ABB RobotStudio station: Table with target.rsstn

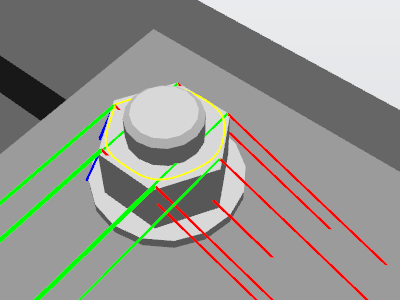
Station Station (saved by RobotStudio 22.3.10141.1)
Controller Controller2
  mechanical unit ROB_1: IRB1410_5_144__01, 6 joints, base frame (0, 0, 0) mm
Layout (positions relative to the parent item):
  - IRB1410_5_144__01 [mechanism, from Robots\IRB1410_5_144_G_01.rslib] at (0, 0, 0) mm; joint values [0.0908, 0.5599, 0.8443, 0.2461, -0.3282, -0.188] (rad or m)
  - table_and_fixture_140 [part, from Training Objects\propeller_table.rslib] at (988.94, -175, 0) mm
  - MyTool [mechanism, from Training Objects\myTool.rslib] at (1105.96, 94, 482.36) mm, rotated rx -180 ry 60 rz -180 deg
Attachment: MyTool is attached to IRB1410_5_144__01 / Link6
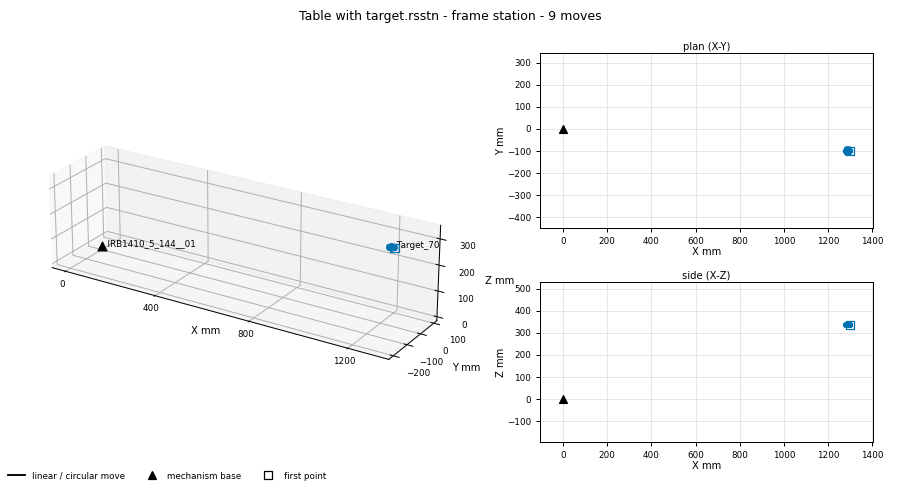
[picture p0: tool path of Table with target.rsstn in frame station, 9 of 9 moves have a stored position in this frame; points joined in program order, loops and branches not executed]
Targets, tools, work objects and paths stored in the station, written as RAPID:
! task T_ROB1
MODULE CalibData
  PERS tooldata MyTool:=[TRUE,[[31.792631019,0,229.638935148],[0.945518576,0,0.325568154,0]],[1,[0,0,1],[1,0,0,0],0,0,0]];
ENDMODULE

! task T_ROB1
MODULE Module1
  CONST robtarget Target_10:=[[1298.606015149,-99.322390924,335.126988795],[0.190805431,0.000000001,0.981627876,0.000000016],[-1,-1,0,0],[9E+09,9E+09,9E+09,9E+09,9E+09,9E+09]];
  CONST robtarget Target_20:=[[1293.833975411,-108.714296883,335.239098516],[0.190804964,0.000000002,0.981627967,0.000000016],[-1,-1,0,0],[9E+09,9E+09,9E+09,9E+09,9E+09,9E+09]];
  CONST robtarget Target_30:=[[1284.016020613,-108.714289941,335.239098112],[0.190804966,0.000000002,0.981627967,0.000000018],[-1,-1,0,0],[9E+09,9E+09,9E+09,9E+09,9E+09,9E+09]];
  CONST robtarget Target_40:=[[1279.428931768,-100.958795352,335.762694702],[0.190804233,-0.000000006,0.981628109,0.000000021],[-1,-1,0,0],[9E+09,9E+09,9E+09,9E+09,9E+09,9E+09]];
  CONST robtarget Target_50:=[[1283.537033031,-91.620253829,335.518813965],[0.190803558,-0.000000004,0.98162824,0.000000021],[-1,-1,0,0],[9E+09,9E+09,9E+09,9E+09,9E+09,9E+09]];
  CONST robtarget Target_60:=[[1294.005032162,-91.620223471,335.518784086],[0.190803449,-0.00000001,0.981628262,0.000000019],[-1,-1,0,0],[9E+09,9E+09,9E+09,9E+09,9E+09,9E+09]];
  CONST robtarget Target_70:=[[1298.231019066,-99.09634302,335.381807422],[0.190802844,-0.000000002,0.981628379,0.000000022],[-1,-1,0,0],[9E+09,9E+09,9E+09,9E+09,9E+09,9E+09]];
  CONST robtarget Target_80:=[[1149.214016226,-99.396362417,334.688483645],[0.190802436,0.000000002,0.981628458,0.00000001],[-1,-1,0,0],[9E+09,9E+09,9E+09,9E+09,9E+09,9E+09]];
  CONST robtarget Target_90:=[[1145.478014256,-109.561191739,336.457915979],[0.190801851,0.000000021,0.981628572,0.000000029],[-1,-1,0,0],[9E+09,9E+09,9E+09,9E+09,9E+09,9E+09]];
  CONST robtarget Target_100:=[[1135.375026076,-109.561186391,336.457899307],[0.190801736,0.000000023,0.981628594,0.000000031],[-1,-1,0,0],[9E+09,9E+09,9E+09,9E+09,9E+09,9E+09]];
  CONST robtarget Target_110:=[[1133.568994915,-109.561194497,334.542287058],[0.190801322,0.000000006,0.981628675,0.000000032],[-1,-1,0,0],[9E+09,9E+09,9E+09,9E+09,9E+09,9E+09]];
  CONST robtarget Target_120:=[[1127.742071524,-109.561197718,324.034410923],[0.190801162,-0.000000004,0.981628706,0.000000029],[-1,-1,0,0],[9E+09,9E+09,9E+09,9E+09,9E+09,9E+09]];
  CONST robtarget Target_130:=[[1132.673969986,-109.561195422,311.197484975],[0.190800844,-0.000000005,0.981628768,0.000000029],[-1,-1,0,0],[9E+09,9E+09,9E+09,9E+09,9E+09,9E+09]];
  CONST robtarget Target_140:=[[1145.380019716,-109.561193614,311.197478936],[0.190800742,-0.000000004,0.981628788,0.000000031],[-1,-1,0,0],[9E+09,9E+09,9E+09,9E+09,9E+09,9E+09]];
  CONST robtarget Target_150:=[[1144.973996719,91.276514259,335.160802204],[0.19080037,-0.000000004,0.98162886,0.000000025],[0,0,-1,0],[9E+09,9E+09,9E+09,9E+09,9E+09,9E+09]];
  CONST robtarget Target_160:=[[1144.973996719,91.276514259,335.160802204],[0.19080037,-0.000000004,0.98162886,0.000000025],[0,0,-1,0],[9E+09,9E+09,9E+09,9E+09,9E+09,9E+09]];
  CONST robtarget Target_170:=[[1144.973996719,91.276514259,335.160802204],[0.19080037,-0.000000004,0.98162886,0.000000025],[0,0,-1,0],[9E+09,9E+09,9E+09,9E+09,9E+09,9E+09]];
  CONST robtarget Target_180:=[[1128.543957252,99.999996916,334.999995635],[0.190800354,-0.000000004,0.981628863,0.000000023],[0,0,-1,0],[9E+09,9E+09,9E+09,9E+09,9E+09,9E+09]];
  CONST robtarget Target_190:=[[1133.739957557,108.999993345,335.000022744],[0.190800372,-0.000000004,0.98162886,0.000000023],[0,0,-1,0],[9E+09,9E+09,9E+09,9E+09,9E+09,9E+09]];
  CONST robtarget Target_200:=[[1144.935946559,99.999995513,322.999995269],[0.190800348,-0.000000005,0.981628864,0.00000002],[0,0,-1,0],[9E+09,9E+09,9E+09,9E+09,9E+09,9E+09]];
  CONST robtarget Target_210:=[[1144.935946559,99.999995513,322.999995269],[0.190800348,-0.000000005,0.981628864,0.00000002],[0,0,-1,0],[9E+09,9E+09,9E+09,9E+09,9E+09,9E+09]];
  CONST robtarget Target_220:=[[1144.935946559,99.999995513,322.999995269],[0.190800348,-0.000000005,0.981628864,0.00000002],[0,0,-1,0],[9E+09,9E+09,9E+09,9E+09,9E+09,9E+09]];
  CONST robtarget Target_230:=[[1144.935946559,99.999995513,322.999995269],[0.190800348,-0.000000005,0.981628864,0.00000002],[0,0,-1,0],[9E+09,9E+09,9E+09,9E+09,9E+09,9E+09]];
  CONST robtarget Target_240:=[[1288.93601006,99.999997691,323.000031211],[0.190800365,-0.000000006,0.981628861,0.00000002],[0,0,-1,0],[9E+09,9E+09,9E+09,9E+09,9E+09,9E+09]];
  CONST robtarget Target_250:=[[1283.740026893,108.999993782,335.000013928],[0.190800047,-0.000000017,0.981628923,0.00000001],[0,0,-1,0],[9E+09,9E+09,9E+09,9E+09,9E+09,9E+09]];
  CONST robtarget Target_260:=[[1294.131991756,109.00000419,335.000026953],[0.190799932,-0.000000024,0.981628945,0.000000011],[0,0,-1,0],[9E+09,9E+09,9E+09,9E+09,9E+09,9E+09]];
  CONST robtarget Target_270:=[[1283.740050918,90.999997159,334.999998956],[0.190799836,-0.000000028,0.981628964,0.000000009],[0,0,-1,0],[9E+09,9E+09,9E+09,9E+09,9E+09,9E+09]];
  CONST robtarget Target_280:=[[1299.327960182,99.999993784,335.00000076],[0.19079964,-0.000000025,0.981629002,0.000000006],[0,0,-1,0],[9E+09,9E+09,9E+09,9E+09,9E+09,9E+09]];
  CONST robtarget Target_290:=[[1288.936033249,93.999995203,340.000015474],[0.190799462,-0.000000027,0.981629036,0.000000004],[0,0,-1,0],[9E+09,9E+09,9E+09,9E+09,9E+09,9E+09]];
  PROC Path_10()
    MoveL Target_70,v1000,z100,MyTool\WObj:=wobj0;
    MoveL Target_70,v1000,z100,MyTool\WObj:=wobj0;
    MoveL Target_10,v1000,z100,MyTool\WObj:=wobj0;
    MoveL Target_20,v1000,z100,MyTool\WObj:=wobj0;
    MoveL Target_30,v1000,z100,MyTool\WObj:=wobj0;
    MoveL Target_40,v1000,z100,MyTool\WObj:=wobj0;
    MoveL Target_50,v1000,z100,MyTool\WObj:=wobj0;
    MoveL Target_60,v1000,z100,MyTool\WObj:=wobj0;
    MoveL Target_70,v1000,z100,MyTool\WObj:=wobj0;
  ENDPROC
ENDMODULE

